// TIA Portal project "Temparature Monitoring and Motor Control Using plc" (V18)

(* hardware
DEVICE "S7-1200 station_1"  S7-1200 Station
   slot 0: "Rack_0"  S7-1200 Rack  Rack  V1.0
   slot 1: "PLC_1"  CPU 1215C DC/DC/DC  6ES7 215-1AG40-0XB0  V4.4
DEVICE "HMI_1"  KTP400 Basic PN
   slot 0: "HMI_1"  KTP400 Basic PN  6AV2 123-2DB03-0AX0  17.0.0.0
   slot 1: "HMI_RT_1"  KTP400 Basic PN  6AV2 123-2DB03-0AX0  17.0.0.0
   slot 5: "HMI_1.IE_CP_1"  PROFINET Interface  17.0.0.0
      slot 1: "PROFINET Interface_1"  PROFINET Interface
         slot 1: "Port_1"  Port
*)

// ===== PLC "PLC_1"  CPU 1215C DC/DC/DC =====

VAR_GLOBAL   // PLC tag table "Default tag table"
   "Motor RV" AT %Q0.1 : Bool;
   "Tag_1" AT %IW64 : Word;
   "Tag_2" AT %MD200 : Real;
   "Temp _Output" AT %MD204 : Real;
   "Fault Memory" AT %M50.5 : Bool;
END_VAR

VAR_GLOBAL   // PLC tag table "System Memory"
   "System Memory" AT %M100.0 : Bool;
END_VAR

VAR_GLOBAL   // PLC tag table "Outputs"
   "Motor Forward" AT %Q0.0 : Bool;
   "15 Hz" AT %Q0.2 : Bool;
   "25 Hz" AT %Q0.3 : Bool;
   "40 Hz" AT %Q0.4 : Bool;
END_VAR

VAR_GLOBAL   // PLC tag table "Inputs"
   "Emergency Stop PB" AT %I0.0 : Bool;
   "Stop Pb" AT %I0.1 : Bool;
   "Start PB" AT %I0.2 : Bool;
   "Motor Run Status (Run_sts)" AT %I0.3 : Bool;
   "Limit switch" AT %I0.4 : Bool;
   "Stop for HMI" AT %M0.5 : Bool;
   "Start for HMI" AT %M0.6 : Bool;
   "Reset PB" AT %I0.7 : Bool;
   "Reset for HMI" AT %M1.0 : Bool;
END_VAR

ORGANIZATION_BLOCK "Main"   // OB1, LAD, ProgramCycle
TITLE = "Main Program Sweep (Cycle)"
{ S7_Optimized_Access := 'TRUE' }
VERSION : 0.1
   VAR_INPUT
      Initial_Call : Bool;   // Initial call of this OB
      Remanence : Bool;   // =True, if remanent data are available
   END_VAR
   VAR_TEMP   // added for the SCL form of the ladder/FBD networks
      _w1 : Bool;
   END_VAR
BEGIN

REGION Network 1
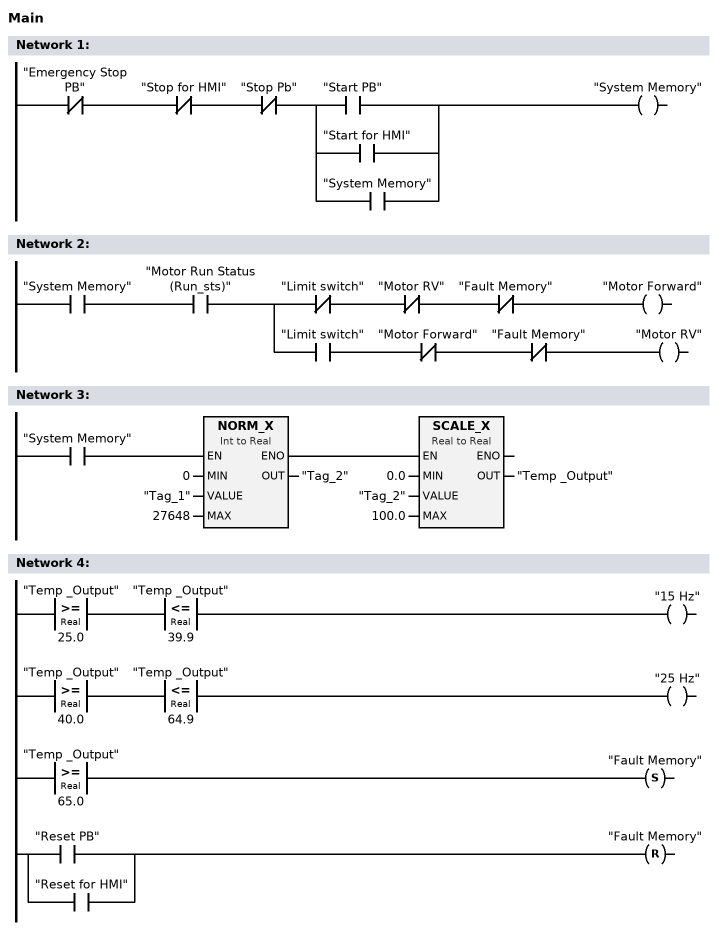
   RUNG wire#powerrail
      I_Contact( "Emergency Stop PB" )
      I_Contact( "Stop for HMI" )
      I_Contact( "Stop Pb" )
      wire#w1
      Contact( "Start PB" )
      wire#w2
      Coil( "System Memory" )
   END_RUNG
   RUNG wire#w1
      Contact( "Start for HMI" )
   END_RUNG wire#w2
   RUNG wire#w1
      Contact( "System Memory" )
   END_RUNG wire#w2
   // the same network as SCL:
   "System Memory" := NOT "Emergency Stop PB" AND NOT "Stop for HMI" AND NOT "Stop Pb" AND ("Start PB" OR "Start for HMI" OR "System Memory");
END_REGION

REGION Network 2
   RUNG wire#powerrail
      Contact( "System Memory" )
      Contact( "Motor Run Status (Run_sts)" )
      wire#w1
      I_Contact( "Limit switch" )
      I_Contact( "Motor RV" )
      I_Contact( "Fault Memory" )
      Coil( "Motor Forward" )
   END_RUNG
   RUNG wire#w1
      Contact( "Limit switch" )
      I_Contact( "Motor Forward" )
      I_Contact( "Fault Memory" )
      Coil( "Motor RV" )
   END_RUNG
   // the same network as SCL:
   #_w1 := "System Memory" AND "Motor Run Status (Run_sts)";
   "Motor Forward" := #_w1 AND NOT "Limit switch" AND NOT "Motor RV" AND NOT "Fault Memory";
   "Motor RV" := #_w1 AND "Limit switch" AND NOT "Motor Forward" AND NOT "Fault Memory";
END_REGION

REGION Network 3
   RUNG wire#powerrail
      Contact( "System Memory" )
      { S7_Templates := "[SrcType := Int, DestType := Real]" } Normalize(min := 0, value := "Tag_1", max := 27648, out => "Tag_2")
      { S7_Templates := "[SrcType := Real, DestType := Real]" } Scale(min := 0.0, value := "Tag_2", max := 100.0, out => "Temp _Output")
   END_RUNG
   // the same network as SCL:
   IF "System Memory" THEN
       "Tag_2" := NORM_X(MIN := 0, VALUE := "Tag_1", MAX := 27648);
       "Temp _Output" := SCALE_X(MIN := 0.0, VALUE := "Tag_2", MAX := 100.0);
   END_IF;
END_REGION

REGION Network 4
   RUNG wire#powerrail
      { S7_Templates := "SrcType := Real" } GE_Contact(in1 := "Temp _Output", in2 := 25.0)
      { S7_Templates := "SrcType := Real" } LE_Contact(in1 := "Temp _Output", in2 := 39.9)
      Coil( "15 Hz" )
   END_RUNG
   RUNG wire#powerrail
      { S7_Templates := "SrcType := Real" } GE_Contact(in1 := "Temp _Output", in2 := 40.0)
      { S7_Templates := "SrcType := Real" } LE_Contact(in1 := "Temp _Output", in2 := 64.9)
      Coil( "25 Hz" )
   END_RUNG
   RUNG wire#powerrail
      { S7_Templates := "SrcType := Real" } GE_Contact(in1 := "Temp _Output", in2 := 65.0)
      S_Coil( "Fault Memory" )
   END_RUNG
   RUNG wire#powerrail
      Contact( "Reset PB" )
      wire#w1
      R_Coil( "Fault Memory" )
   END_RUNG
   RUNG wire#powerrail
      Contact( "Reset for HMI" )
   END_RUNG wire#w1
   // the same network as SCL:
   "15 Hz" := ("Temp _Output" >= 25.0) AND ("Temp _Output" <= 39.9);
   "25 Hz" := ("Temp _Output" >= 40.0) AND ("Temp _Output" <= 64.9);
   IF "Temp _Output" >= 65.0 THEN "Fault Memory" := TRUE; END_IF;
   IF "Reset PB" OR "Reset for HMI" THEN "Fault Memory" := FALSE; END_IF;
END_REGION
END_ORGANIZATION_BLOCK

(* ===== HMI "HMI_RT_1" =====
system functions are stored by id; their names below are inferred from use
connection "HMI_Connection_1": ETHERNET, SMART_S7_1200_OMS

HMI tags "Default tag table"
   "Tag_ScreenNumber" : UInt, internal
   "Stop for HMI" : Bool = PLC "Stop for HMI" AT %M0.5, 1 s
   "Start for HMI" : Bool = PLC "Start for HMI" AT %M0.6, 1 s
   "Reset for HMI" : Bool = PLC "Reset for HMI" AT %M1.0, 1 s
   "Fault Memory" : Bool = PLC "Fault Memory" AT %M50.5, 1 s
   "Motor Forward" : Bool = PLC "Motor Forward" AT %Q0.0, 1 s
   "15 Hz" : Bool = PLC "15 Hz" AT %Q0.2, 1 s
   "25 Hz" : Bool = PLC "25 Hz" AT %Q0.3, 1 s
   "Motor RV" : Bool = PLC "Motor RV" AT %Q0.1, 1 s
   "Temp _Output" : Real = PLC "Temp _Output" AT %MD204, 1 s

Template "Template_1" 480x272
   Button "Exit" at 388,227 size 63x44; TextOff 'Exit'; PictureOff "ExitRuntime_KTP400_Basic_PN_TR"; PictureOn "ExitRuntime_KTP400_Basic_PN_TR"
      on Release: StopRuntime(0)
   Button "Template_Button" at 268,227 size 63x44; TextOff 'Text'
   Button "Alarms" at 148,227 size 63x44; TextOff 'Alarms'; PictureOff "AlarmDisplay_KTP400_Basic_PN_TR"; PictureOn "AlarmDisplay_KTP400_Basic_PN_TR"
      on Release: function_ef3f5d25("Alarm window_Unacknowledged", -1)
   Button "Start screen" at 28,227 size 63x44; TextOff 'Start screen'; PictureOff "NavigateHome_KTP400_Basic_PN_TR"; PictureOn "NavigateHome_KTP400_Basic_PN_TR"
      on Release: ActivateScreen("Root screen", 0)
   SymbolicIOField "Symbolic_IO_Field_Screen" at 82,8 size 311x29; TextOff '0'; TextOn '1'; TextList "TextList_ScreenNames"
      ProcessValue <- "Tag_ScreenNumber"
      on Change: ActivateScreenByNumber("Tag_ScreenNumber", 0)
   DateTimeField "HmiScreenItemData" at 395,22 size 85x22
   DateTimeField "HmiScreenItemData_1" at 395,0 size 85x22
   GraphicView "Logo" at 0,0 size 80x45; Picture "Logo of HMI_1"

screen "Root screen" 480x272, template "Template_1"
   on GenerateScreen: SetTag("Tag_ScreenNumber", 1)
   GraphicView "Graphic view_1" at 0,0 size 480x272; Picture "wallpaperbetter (1)"
   TextField "Text field_1" at 60,16 size 275x20; Text 'Temparature Monitoring & Motor Control'
   Button "Button_1" at 52,95 size 63x35; TextOff 'Stop'
      on Press: function_b14e0dd5("Stop for HMI", 0)
   Button "Button_2" at 52,145 size 63x35; TextOff 'Start'
      on Press: function_b14e0dd5("Start for HMI", 0)
   Circle "Circle_1" at 52,201 size 47x47
      Visibility <- "Motor Forward"
      Appearance <- "Motor Forward"
   TextField "Text field_2" at 46,249 size 61x20; Text 'Motor FW'
   TextField "Text field_3" at 142,248 size 38x20; Text '15 HZ'
   Circle "Circle_3" at 220,201 size 47x47
      Appearance <- "25 Hz"
   TextField "Text field_4" at 220,248 size 37x20; Text '25 Hz'
   Circle "Circle_4" at 303,200 size 47x47
      Appearance <- "Motor RV"
   TextField "Text field_5" at 297,248 size 60x22; Text 'Motor RV'
   IOField "I/O field_1" at 384,143 size 96x32; FormatPattern 999
      ProcessValue <- "Temp _Output"
   Button "Button_3" at 137,120 size 63x35; TextOff 'Reset'
      on Press: function_b14e0dd5("Reset for HMI", 0)
   GraphicView "Graphic view_2" at 47,13 size 370x221; Picture "Graphic_1"
      Visibility <- "Fault Memory"
      Appearance <- "15 Hz"
*)